(* PLC project int2real_conversion, Dassault Systèmes ControlBuild 2024x *)
(* stored: creationDateTime 2023-10-03T11:13:30-01:00 *)

(* This module converts an integer input into a real output. *)
FUNCTION_BLOCK equipment_library.int2real_conversion
  VAR_INPUT
    dintInput : DINT := 0;
    intInput : INT := 0;
  END_VAR
  VAR_OUTPUT
    output : REAL := 0.0;
  END_VAR
  VAR CONSTANT
    selectDouble : BOOL := true;
  END_VAR


ACTION C_source_code:
/* ----------------------------------------------------------------	*/
/* Type : Model of Operative Behaviour					*/
/* Category :  Toolbox							*/
/* Author : Dassault Systemes						*/
/* Update date : June 2018						*/
/* ----------------------------------------------------------------	*/
/* This module converts an integer dintInput into a real output.	*/
/*										*/
/* The parameter allows to switch between the DINT input (true by	*/
/* default) or the INT input (false)
/* ----------------------------------------------------------------	*/

if (selectDouble)  output = dintInput;
else output = intInput;
END_ACTION
END_FUNCTION_BLOCK
